// TIA Portal V18 export
DATA_BLOCK "Function Metering pgm"   // DB41
{ S7_Optimized_Access := 'TRUE' }
VERSION : 0.1
// stored: AutoNumber true, DBAccessibleFromOPCUA true, IsOnlyStoredInLoadMemory false, IsRetainMemResEnabled false, IsWriteProtectedInAS false, MemoryReserve 100
   VAR RETAIN
      input : Struct
         "Set Flowrate" : Real;
         "Set time" : DInt;
         "Flowrate adjustment A" : Real;
         "Flowrate adjustment B" : Real;
         "set qty" : Real;
      END_STRUCT;
   END_VAR
   VAR
      Control : Struct
         "Start metering" : Bool;
         "Do continuous metering" : Bool;
         "Stop metering" : Bool;
         "metering running" : Bool;
         "metering completed" : Bool;
      END_STRUCT;
      output : Struct
         "ON_pump A" : Bool;
         "ON_pump B" : Bool;
         ON_mixer : Bool;
         "ON_outlet Valve A" : Bool;
         "Running time" : Int;
         "ON_outlet valve B" : Bool;
         "Volume dispensed" : Real;
         "ON_inlet A" : Bool;
         "ON_inlet B" : Bool;
      END_STRUCT;
   END_VAR
BEGIN
END_DATA_BLOCK
